FUNCTION_BLOCK MERGE2_WITH_QUEUE
  (* Version 1.0, 2005-12-27, Oscar Ljungkrantz, Chalmers *)
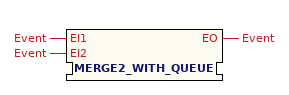
  EVENT_INPUT
    EI1;
    EI2;
  END_EVENT
  EVENT_OUTPUT
    EO;
  END_EVENT
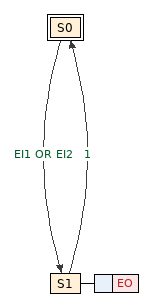
  EC_STATES
    S0;
    S1 : -> EO;
  END_STATES
  EC_TRANSITIONS
    S0 TO S1 := EI1 OR EI2;
    S1 TO S0 := 1;
  END_TRANSITIONS
END_FUNCTION_BLOCK
(* other elements stored in the file *)
(* ECState Name="S2"> <ECAction Output="EO" /> <ECAction Output="EO" /> </ECState *)
(* ECTransition Source="S0" Destination="S1" Condition="(EI1 AND NOT EI2) OR (EI2 AND NOT EI1)" /> <ECTransition Source="S0" Destination="S2" Condition="EI1 AND EI2" /> <ECTransition Source="S1" Destination="S2" Condition="EI1 AND EI2" /> <ECTransition Source="S1" Destination="S1" Condition="(EI1 AND NOT EI2) OR (EI2 AND NOT EI1)" /> <ECTransition Source="S1" Destination="S0" Condition="NOT EI1 AND NOT EI2" /> <ECTransition Source="S2" Destination="S2" Condition="EI1 AND EI2" /> <ECTransition Source="S2" Destination="S1" Condition="(EI1 AND NOT EI2) OR (EI2 AND NOT EI1)" /> <ECTransition Source="S2" Destination="S0" Condition="NOT EI1 AND NOT EI2" / *)
